DATA_BLOCK "Lifter.Encoder_DB"
{ S7_Optimized_Access := 'TRUE' }
VERSION : 0.1
NON_RETAIN
"Encoder_ELAP"

BEGIN

END_DATA_BLOCK

